FUNCTION_BLOCK Sequenz_1 EXTENDS FB_Basis IMPLEMENTS I_Sequenz
VAR_INPUT
	// Benötigter Skill
	Move_2P2		:I_Skill_Roboter;
	Gripper			:I_Skill_Greifer;
	
	// Benötigte Parameter
	Position_1		:sRoboterProzessVariablen;
	Position_2		:sRoboterProzessVariablen;
	GreifPos_1		:sSmartGreiferProzessVariablen;
	GreifPos_2		:sSmartGreiferProzessVariablen;
END_VAR
VAR_OUTPUT
END_VAR
VAR
END_VAR

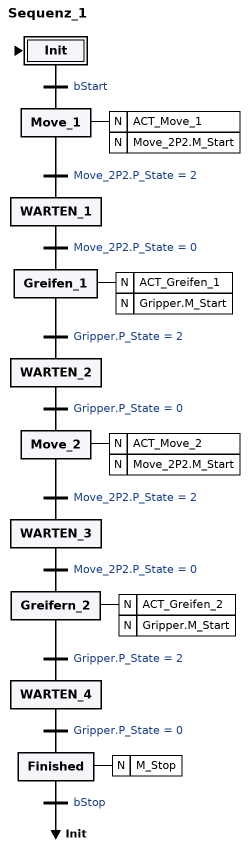
INITIAL_STEP Init:
END_STEP
TRANSITION FROM Init TO Move_1
    := bStart;
END_TRANSITION
STEP Move_1:
    ACT_Move_1(N);
    Move_2P2.M_Start(N);
END_STEP
TRANSITION FROM Move_1 TO WARTEN_1
    := Move_2P2.P_State = 2;
END_TRANSITION
STEP WARTEN_1:
END_STEP
TRANSITION FROM WARTEN_1 TO Greifen_1
    := Move_2P2.P_State = 0;
END_TRANSITION
STEP Greifen_1:
    ACT_Greifen_1(N);
    Gripper.M_Start(N);
END_STEP
TRANSITION FROM Greifen_1 TO WARTEN_2
    := Gripper.P_State = 2;
END_TRANSITION
STEP WARTEN_2:
END_STEP
TRANSITION FROM WARTEN_2 TO Move_2
    := Gripper.P_State = 0;
END_TRANSITION
STEP Move_2:
    ACT_Move_2(N);
    Move_2P2.M_Start(N);
END_STEP
TRANSITION FROM Move_2 TO WARTEN_3
    := Move_2P2.P_State = 2;
END_TRANSITION
STEP WARTEN_3:
END_STEP
TRANSITION FROM WARTEN_3 TO Greifern_2
    := Move_2P2.P_State = 0;
END_TRANSITION
STEP Greifern_2:
    ACT_Greifen_2(N);
    Gripper.M_Start(N);
END_STEP
TRANSITION FROM Greifern_2 TO WARTEN_4
    := Gripper.P_State = 2;
END_TRANSITION
STEP WARTEN_4:
END_STEP
TRANSITION FROM WARTEN_4 TO Finished
    := Gripper.P_State = 0;
END_TRANSITION
STEP Finished:
    M_Stop(N);
END_STEP
TRANSITION FROM Finished TO Init
    := bStop;
END_TRANSITION

ACTION ACT_Greifen_1:
Gripper.P_Prozessparameter := GreifPos_1;
END_ACTION

ACTION ACT_Greifen_2:
Gripper.P_Prozessparameter := GreifPos_2;
END_ACTION

ACTION ACT_Move_1:
Move_2P2.P_Prozessparameter := Position_1;
END_ACTION

ACTION ACT_Move_2:
Move_2P2.P_Prozessparameter := Position_2;
END_ACTION

END_FUNCTION_BLOCK

(* stored: Version 1.1.0.1
   POU Sequenz_1: Id {507cb58e-3ca6-42f6-81f1-24566c69ed33}, SpecialFunc None
   Folder 01_Zuweisung: Id {b5adafe3-e7fb-411f-abc4-8082512de09d}
   Action ACT_Greifen_1: Id {c3347e58-9deb-474d-9006-43a59c6d0690}
   Action ACT_Greifen_2: Id {d1826670-5996-45fb-9870-bd7b6932d4e3}
   Action ACT_Move_1: Id {3bfceb9a-3a7f-424e-8a95-533c78d8d8bf}
   Action ACT_Move_2: Id {10b6fe2f-3786-4b6f-96b2-58ba58bf6d37} *)
